// TIA Portal V20 export
DATA_BLOCK "Alarms"   // DB150
// stored: MemoryReserve 100, Namespace Unit1.Em0
   VAR
      emAlarms { ExternalWritable := 'False'} : "LAF_typeAlarms";
      maintenanceFaults { ExternalWritable := 'False'} : Array[0..199] of Bool;   // PFE Maintenance Faults
      productionFaults { ExternalWritable := 'False'} : Array[0..199] of Bool;   // PFE Production Faults
      toolingFault { ExternalWritable := 'False'} : Array[0..199] of Bool;   // PFE Tooling Faults
      qualityFault { ExternalWritable := 'False'} : Array[0..199] of Bool;   // PFE Quality Faults
      throughputFaultBlocked { ExternalWritable := 'False'} : Array[0..199] of Bool;   // PFE Throughput Fault Blocked
      throughputFaultStarved { ExternalWritable := 'False'} : Array[0..199] of Bool;   // PFE Throughput Fault Starved
      throughputFault { ExternalWritable := 'False'} : Array[0..199] of Bool;   // PFE Throughput Fault
      systemFaultGeneral { ExternalWritable := 'False'} : Array[0..199] of Bool;   // PFE System Fault General
      materialFault { ExternalWritable := 'False'} : Array[0..199] of Bool;   // PFE Material Fault
      maintenanceWarnings { ExternalWritable := 'False'} : Array[0..199] of Bool;   // PFE Maintenance Warnings
      productionWarning { ExternalWritable := 'False'} : Array[0..199] of Bool;   // PFE Production Warning
      toolingWarning { ExternalWritable := 'False'} : Array[0..199] of Bool;   // PFE Tooling Warning
      qualityWarning { ExternalWritable := 'False'} : Array[0..199] of Bool;   // PFE Quality Warning
      throughputWarning { ExternalWritable := 'False'} : Array[0..199] of Bool;   // PFE Throughput Warning
      systemWarning { ExternalWritable := 'False'} : Array[0..199] of Bool;   // PFE System Warning
      materialWarning { ExternalWritable := 'False'} : Array[0..199] of Bool;   // PFE Material Warning
      maintenanceStatus { ExternalWritable := 'False'} : Array[0..199] of Bool;   // PFE Maintenance Status
      productionStatus { ExternalWritable := 'False'} : Array[0..199] of Bool;   // PFE Production Status
      toolingStatus { ExternalWritable := 'False'} : Array[0..199] of Bool;   // PFE Tooling Status
      qualityStatus { ExternalWritable := 'False'} : Array[0..199] of Bool;   // PFE Quality Status
      throughputStatus { ExternalWritable := 'False'} : Array[0..199] of Bool;   // PFE Throughput Status
      systemStatus { ExternalWritable := 'False'} : Array[0..199] of Bool;   // PFE System Status
      materialStatus { ExternalWritable := 'False'} : Array[0..199] of Bool;   // PFE Material Status
      TonMaintenanceFault { ExternalWritable := 'False'} : Array[0..199] of TON_TIME;   // PFE Maintenance Faults Ton Timer
      TonProductionFault { ExternalWritable := 'False'} : Array[0..199] of TON_TIME;   // PFE Production Faults Ton Timer
      TonToolingFault { ExternalWritable := 'False'} : Array[0..199] of TON_TIME;   // PFE Tooling Faults Ton Timer
      TonQualityFault { ExternalWritable := 'False'} : Array[0..199] of TON_TIME;   // PFE Quality Faults Ton Timer
      TonThroughputFaultBlocked { ExternalWritable := 'False'} : Array[0..199] of TON_TIME;   // PFE Throughput Fault Blocked Ton Timer
      TonThroughputFaultStarved { ExternalWritable := 'False'} : Array[0..199] of TON_TIME;   // PFE Throughput Fault Starved Ton Timer
      TonThroughputFault { ExternalWritable := 'False'} : Array[0..199] of TON_TIME;   // PFE Throughput Fault Ton Timer
      TonSystemFaultGeneral { ExternalWritable := 'False'} : Array[0..199] of TON_TIME;   // PFE System Fault General Ton Timer
      TonMaterialFault { ExternalWritable := 'False'} : Array[0..199] of TON_TIME;   // PFE Material Fault Ton Timer
      TonMaintenanceWarning { ExternalWritable := 'False'} : Array[0..199] of TON_TIME;   // PFE Maintenance Warnings Ton Timer
      TonProductionWarning { ExternalWritable := 'False'} : Array[0..199] of TON_TIME;   // PFE Production Warning Ton Timer
      TonToolingWarning { ExternalWritable := 'False'} : Array[0..199] of TON_TIME;   // PFE Tooling Warning Ton Timer
      TonQualityWarning { ExternalWritable := 'False'} : Array[0..199] of TON_TIME;   // PFE Quality Warning Ton Timer
      TonThroughputWarning { ExternalWritable := 'False'} : Array[0..199] of TON_TIME;   // PFE Throughput Warning Ton Timer
      TonSystemWarning { ExternalWritable := 'False'} : Array[0..199] of TON_TIME;   // PFE System Warning Ton Timer
      TonMaterialWarning { ExternalWritable := 'False'} : Array[0..199] of TON_TIME;   // PFE Material Warning Ton Timer
      TonMaintenanceStatus { ExternalWritable := 'False'} : Array[0..199] of TON_TIME;   // PFE Maintenance Status Ton Timer
      TonProductionStatus { ExternalWritable := 'False'} : Array[0..199] of TON_TIME;   // PFE Production Status Ton Timer
      TonToolingStatus { ExternalWritable := 'False'} : Array[0..199] of TON_TIME;   // PFE Tooling Status Ton Timer
      TonQualityStatus { ExternalWritable := 'False'} : Array[0..199] of TON_TIME;   // PFE Quality Status Ton Timer
      TonThroughputStatus { ExternalWritable := 'False'} : Array[0..199] of TON_TIME;   // PFE Throughput Status Ton Timer
      TonSystemStatus { ExternalWritable := 'False'} : Array[0..199] of TON_TIME;   // PFE System Status Ton Timer
      TonMaterialStatus { ExternalWritable := 'False'} : Array[0..199] of TON_TIME;   // PFE Material Status Ton Timer
   END_VAR
BEGIN
   // maintenanceFaults[0] : RFID Error
   // maintenanceFaults[1] : Em0 Homed Time Over
   // productionFaults[0] : Tension not established
   // productionFaults[1] : Roll Change Box key not in AUTO position
   // materialFault[0] : Material Depleted
END_DATA_BLOCK
